ABB RobotStudio station: Solution4Laboratorio2_4.rsstn

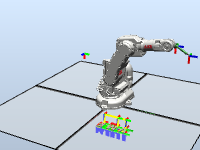
Station Solution4Laboratorio2_4 (saved by RobotStudio 6.8.8307.1040)
Controller IRB_140_6kg_0.81m
  mechanical unit ROB_1: IRB140_6_81_C_03, 6 joints, base frame (0, 0, 0) mm
Layout (positions relative to the parent item):
  - IRB140_6_81_C_03 [mechanism, from Robots\IRB140_6_81_C_G_03.rslib] at (0, 0, 0) mm; joint values [1.5708, 0.4306, -0.6009, 0, 0.1703, 0] (rad or m)
  - Modelo [graphiccomponentgroup] at (0, 659.78, 743.53) mm, rotated rx 90 ry 0 rz 180 deg
    - Component1:1 [part] at (0, -4, 6.93) mm
    - Component2:1 [part] at (0, 0, 0) mm
    - Component3:1 [part] at (0, 0, 0) mm
    - marcador v3:1 [part] at (0, -12.99, 28.51) mm, rotated rx 30 ry 0 rz 0 deg
  - INICIALES3 v2 [part] at (400, 400, 0) mm, rotated rx 0 ry 0 rz -90 deg
Attachment: Modelo is attached to IRB140_6_81_C_03 / Link6
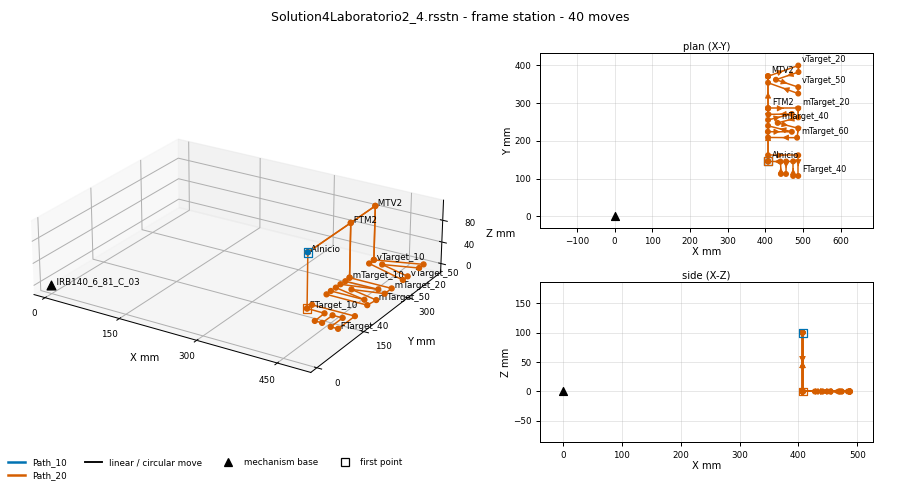
[picture p0: tool path of Solution4Laboratorio2_4.rsstn in frame station, 40 of 42 moves have a stored position in this frame; points joined in program order, loops and branches not executed]
Targets, tools, work objects and paths stored in the station, written as RAPID:
! task T_ROB1
MODULE CalibData
  TASK PERS wobjdata Workobject_INICIALES:=[FALSE,TRUE,"",[[407.13,371.405,0],[0,0,1,0]],[[0,0,0],[1,0,0,0]]];
  TASK PERS tooldata Tooldata_MARCADOR:=[TRUE,[[74.149,0,131.75],[1,0,0,0]],[0.06,[0,0,70],[1,0,0,0],0,0,0]];
ENDMODULE

! task T_ROB1
MODULE Module1
  CONST robtarget vTarget_10:=[[0.326,-0.089,0],[1,0,0,0],[0,0,0,0],[9E+09,9E+09,9E+09,9E+09,9E+09,9E+09]];
  CONST robtarget vTarget_20:=[[-80.066,28.469,0],[1,0,0,0],[0,0,0,0],[9E+09,9E+09,9E+09,9E+09,9E+09,9E+09]];
  CONST robtarget vTarget_30:=[[-80.616,11.146,0],[1,0,0,0],[0,0,0,0],[9E+09,9E+09,9E+09,9E+09,9E+09,9E+09]];
  CONST robtarget vTarget_40:=[[-20.791,-9.168,0],[1,0,0,0],[0,0,0,0],[9E+09,9E+09,9E+09,9E+09,9E+09,9E+09]];
  CONST robtarget vTarget_50:=[[-80,-28.758,0],[1,0,0,0],[0,0,0,0],[9E+09,9E+09,9E+09,9E+09,9E+09,9E+09]];
  CONST robtarget vTarget_60:=[[-80,-45.893,0],[1,0,0,0],[0,0,0,0],[9E+09,9E+09,9E+09,9E+09,9E+09,9E+09]];
  CONST robtarget vTarget_70:=[[0,-17.244,0],[1,0,0,0],[0,0,0,0],[9E+09,9E+09,9E+09,9E+09,9E+09,9E+09]];
  CONST robtarget mTarget_10:=[[0,-84.966,0],[1,0,0,0],[0,0,0,0],[9E+09,9E+09,9E+09,9E+09,9E+09,9E+09]];
  CONST robtarget mTarget_20:=[[-80,-84.966,0],[1,0,0,0],[0,0,0,0],[9E+09,9E+09,9E+09,9E+09,9E+09,9E+09]];
  CONST robtarget mTarget_30:=[[-80,-109.14,0],[1,0,0,0],[0,0,0,0],[9E+09,9E+09,9E+09,9E+09,9E+09,9E+09]];
  CONST robtarget mTarget_40:=[[-25.429,-123.656,0],[1,0,0,0],[0,0,0,0],[9E+09,9E+09,9E+09,9E+09,9E+09,9E+09]];
  CONST robtarget mTarget_50:=[[-80,-138.008,0],[1,0,0,0],[0,0,0,0],[9E+09,9E+09,9E+09,9E+09,9E+09,9E+09]];
  CONST robtarget mTarget_60:=[[-76.954,-162.904,0],[1,0,0,0],[0,0,0,0],[9E+09,9E+09,9E+09,9E+09,9E+09,9E+09]];
  CONST robtarget mTarget_70:=[[0,-162.237,0],[1,0,0,0],[0,0,0,0],[9E+09,9E+09,9E+09,9E+09,9E+09,9E+09]];
  CONST robtarget mTarget_80:=[[0.53,-147.013,0],[1,0,0,0],[0,0,0,0],[9E+09,9E+09,9E+09,9E+09,9E+09,9E+09]];
  CONST robtarget mTarget_90:=[[-62.974,-147.23,0],[1,0,0,0],[0,0,0,0],[9E+09,9E+09,9E+09,9E+09,9E+09,9E+09]];
  CONST robtarget mTarget_100:=[[0,-131.35,0],[1,0,0,0],[0,0,0,0],[9E+09,9E+09,9E+09,9E+09,9E+09,9E+09]];
  CONST robtarget mTarget_110:=[[0,-115.798,0],[1,0,0,0],[0,0,0,0],[9E+09,9E+09,9E+09,9E+09,9E+09,9E+09]];
  CONST robtarget mTarget_120:=[[-62.974,-99.973,0],[1,0,0,0],[0,0,0,0],[9E+09,9E+09,9E+09,9E+09,9E+09,9E+09]];
  CONST robtarget mTarget_130:=[[-0.986,-101.003,0],[1,0,0,0],[0,0,0,0],[9E+09,9E+09,9E+09,9E+09,9E+09,9E+09]];
  CONST robtarget FTarget_10:=[[0,-225.593,0],[1,0,0,0],[0,0,0,0],[9E+09,9E+09,9E+09,9E+09,9E+09,9E+09]];
  CONST robtarget FTarget_20:=[[0,-209.44,0],[1,0,0,0],[0,0,0,0],[9E+09,9E+09,9E+09,9E+09,9E+09,9E+09]];
  CONST robtarget FTarget_30:=[[-80,-209.44,0],[1,0,0,0],[0,0,0,0],[9E+09,9E+09,9E+09,9E+09,9E+09,9E+09]];
  CONST robtarget FTarget_40:=[[-80,-264.284,0],[1,0,0,0],[0,0,0,0],[9E+09,9E+09,9E+09,9E+09,9E+09,9E+09]];
  CONST robtarget FTarget_50:=[[-66.466,-264.284,0],[1,0,0,0],[0,0,0,0],[9E+09,9E+09,9E+09,9E+09,9E+09,9E+09]];
  CONST robtarget FTarget_60:=[[-66.466,-225.593,0],[1,0,0,0],[0,0,0,0],[9E+09,9E+09,9E+09,9E+09,9E+09,9E+09]];
  CONST robtarget FTarget_70:=[[-47.849,-225.879,0],[1,0,0,0],[0,0,0,0],[9E+09,9E+09,9E+09,9E+09,9E+09,9E+09]];
  CONST robtarget FTarget_80:=[[-47.53,-258.99,0],[1,0,0,0],[0,0,0,0],[9E+09,9E+09,9E+09,9E+09,9E+09,9E+09]];
  CONST robtarget FTarget_90:=[[-33.997,-258.99,0],[1,0,0,0],[0,0,0,0],[9E+09,9E+09,9E+09,9E+09,9E+09,9E+09]];
  CONST robtarget FTarget_100:=[[-33.164,-226.306,0],[1,0,0,0],[0,0,0,0],[9E+09,9E+09,9E+09,9E+09,9E+09,9E+09]];
  CONST robtarget AInicio:=[[0,-225.593,-100],[1,0,0,0],[0,0,0,0],[9E+09,9E+09,9E+09,9E+09,9E+09,9E+09]];
  CONST robtarget FTM2:=[[0,-84.966,-100],[1,0,0,0],[0,0,0,0],[9E+09,9E+09,9E+09,9E+09,9E+09,9E+09]];
  CONST robtarget MTV2:=[[0.326,-0.089,-100],[1,0,0,0],[0,0,0,0],[9E+09,9E+09,9E+09,9E+09,9E+09,9E+09]];
  CONST robtarget ZInicio:=[[0,-225.593,-100],[1,0,0,0],[0,0,0,0],[9E+09,9E+09,9E+09,9E+09,9E+09,9E+09]];
  CONST robtarget FTarget_110:=[[0,-225.593,0],[1,0,0,0],[0,0,0,0],[9E+09,9E+09,9E+09,9E+09,9E+09,9E+09]];
  CONST robtarget mTarget_140:=[[0,-84.966,0],[1,0,0,0],[0,0,0,0],[9E+09,9E+09,9E+09,9E+09,9E+09,9E+09]];
  CONST robtarget vTarget_80:=[[0.326,-0.089,0],[1,0,0,0],[0,0,0,0],[9E+09,9E+09,9E+09,9E+09,9E+09,9E+09]];
  CONST robtarget vTarget_80_final:=[[0.326,-0.089,-100],[1,0,0,0],[0,0,0,0],[9E+09,9E+09,9E+09,9E+09,9E+09,9E+09]];
  CONST robtarget MTV1:=[[0,-84.966,-100],[1,0,0,0],[0,0,0,0],[9E+09,9E+09,9E+09,9E+09,9E+09,9E+09]];
  CONST robtarget FTM1:=[[0,-225.593,-100],[1,0,0,0],[0,0,0,0],[9E+09,9E+09,9E+09,9E+09,9E+09,9E+09]];
  CONST jointtarget HomePosition:=[[0,0,0,0,0,0],[9E+09,9E+09,9E+09,9E+09,9E+09,9E+09]];
  CONST jointtarget ChangeTool:=[[90.000002504,24.671787339,-34.427722191,-0.000016273,9.755934852,0.000016038],[9E+09,9E+09,9E+09,9E+09,9E+09,9E+09]];
  PROC Path_10()
    MoveJ AInicio,v100,z10,Tooldata_MARCADOR\WObj:=Workobject_INICIALES;
  ENDPROC
  PROC Path_20()
    MoveL FTarget_10,v100,z10,Tooldata_MARCADOR\WObj:=Workobject_INICIALES;
    MoveL FTarget_20,v100,z10,Tooldata_MARCADOR\WObj:=Workobject_INICIALES;
    MoveL FTarget_30,v100,z10,Tooldata_MARCADOR\WObj:=Workobject_INICIALES;
    MoveL FTarget_40,v100,z10,Tooldata_MARCADOR\WObj:=Workobject_INICIALES;
    MoveL FTarget_50,v100,z10,Tooldata_MARCADOR\WObj:=Workobject_INICIALES;
    MoveL FTarget_60,v100,z10,Tooldata_MARCADOR\WObj:=Workobject_INICIALES;
    MoveL FTarget_70,v100,z10,Tooldata_MARCADOR\WObj:=Workobject_INICIALES;
    MoveL FTarget_80,v100,z10,Tooldata_MARCADOR\WObj:=Workobject_INICIALES;
    MoveL FTarget_90,v100,z10,Tooldata_MARCADOR\WObj:=Workobject_INICIALES;
    MoveL FTarget_100,v100,z10,Tooldata_MARCADOR\WObj:=Workobject_INICIALES;
    MoveL FTarget_110,v100,z10,Tooldata_MARCADOR\WObj:=Workobject_INICIALES;
    MoveL FTM1,v100,z10,Tooldata_MARCADOR\WObj:=Workobject_INICIALES;
    MoveL FTM2,v100,z10,Tooldata_MARCADOR\WObj:=Workobject_INICIALES;
    MoveL mTarget_10,v100,z10,Tooldata_MARCADOR\WObj:=Workobject_INICIALES;
    MoveL mTarget_20,v100,z10,Tooldata_MARCADOR\WObj:=Workobject_INICIALES;
    MoveL mTarget_30,v100,z10,Tooldata_MARCADOR\WObj:=Workobject_INICIALES;
    MoveL mTarget_40,v100,z10,Tooldata_MARCADOR\WObj:=Workobject_INICIALES;
    MoveL mTarget_50,v100,z10,Tooldata_MARCADOR\WObj:=Workobject_INICIALES;
    MoveL mTarget_60,v100,z10,Tooldata_MARCADOR\WObj:=Workobject_INICIALES;
    MoveL mTarget_70,v100,z10,Tooldata_MARCADOR\WObj:=Workobject_INICIALES;
    MoveL mTarget_80,v100,z10,Tooldata_MARCADOR\WObj:=Workobject_INICIALES;
    MoveL mTarget_90,v100,z10,Tooldata_MARCADOR\WObj:=Workobject_INICIALES;
    MoveL mTarget_100,v100,z10,Tooldata_MARCADOR\WObj:=Workobject_INICIALES;
    MoveL mTarget_110,v100,z10,Tooldata_MARCADOR\WObj:=Workobject_INICIALES;
    MoveL mTarget_120,v100,z10,Tooldata_MARCADOR\WObj:=Workobject_INICIALES;
    MoveL mTarget_130,v100,z10,Tooldata_MARCADOR\WObj:=Workobject_INICIALES;
    MoveL mTarget_140,v100,z10,Tooldata_MARCADOR\WObj:=Workobject_INICIALES;
    MoveL MTV1,v100,z10,Tooldata_MARCADOR\WObj:=Workobject_INICIALES;
    MoveL MTV2,v100,z10,Tooldata_MARCADOR\WObj:=Workobject_INICIALES;
    MoveL vTarget_10,v100,z10,Tooldata_MARCADOR\WObj:=Workobject_INICIALES;
    MoveL vTarget_20,v100,z10,Tooldata_MARCADOR\WObj:=Workobject_INICIALES;
    MoveL vTarget_30,v100,z10,Tooldata_MARCADOR\WObj:=Workobject_INICIALES;
    MoveL vTarget_40,v100,z10,Tooldata_MARCADOR\WObj:=Workobject_INICIALES;
    MoveL vTarget_50,v100,z10,Tooldata_MARCADOR\WObj:=Workobject_INICIALES;
    MoveL vTarget_60,v100,z10,Tooldata_MARCADOR\WObj:=Workobject_INICIALES;
    MoveL vTarget_70,v100,z10,Tooldata_MARCADOR\WObj:=Workobject_INICIALES;
    MoveL vTarget_80,v100,z10,Tooldata_MARCADOR\WObj:=Workobject_INICIALES;
    MoveL vTarget_80_final,v100,z10,Tooldata_MARCADOR\WObj:=Workobject_INICIALES;
    MoveL ZInicio,v100,z10,Tooldata_MARCADOR\WObj:=Workobject_INICIALES;
  ENDPROC
  PROC Home1()
    MoveAbsJ HomePosition,v100,z10,Tooldata_MARCADOR\WObj:=Workobject_INICIALES;
  ENDPROC
  PROC ToolChange()
    MoveAbsJ ChangeTool,v50,z10,Tooldata_MARCADOR\WObj:=Workobject_INICIALES;
  ENDPROC
  PROC main()
    Home1;
    WaitDI EntDI_1,1;
    SetDO SalDO_1,1;
    Path_10;
    Path_20;
    Home1;
    WaitDI EntDI_2,1;
    ToolChange;
    SetDO SalDO_1,0;
  ENDPROC
ENDMODULE

